(* IEC 61131-3 sources: AXOpen/src/components.drives/ctrl/src/AxoDrives (part 3) *)

            IF Enable THEN
                AxoReadActualPosition_Task.SwitchOn();
            ELSE
                AxoReadActualPosition_Task.SwitchOff();
                // THIS.MC_ReadActualPosition(AxisRef, FALSE);
            END_IF;

            Valid       := AxoReadActualPosition_Valid;
            Busy        :=  AxoReadActualPosition_Busy;
            Error       :=  AxoReadActualPosition_Error;
            ErrorID     :=  AxoReadActualPosition_ErrorID;
            Position    := AxoReadActualPosition_Value;

            AxoReadActualPosition  := AxoReadActualPosition_Task;
        END_METHOD

        ///<summary>
        /// This method returns the value of the actual velocity as long as ‘Enable’ is set. ‘Valid’ is true when the
        /// dataoutput ‘Velocity’ is valid. If ‘Enable’ is Reset, the data loses its validity, and all outputs are reset,
        /// no matter if new data is available.
        ///<summary>
        METHOD PUBLIC AxoReadActualVelocity    : IAxoToggleTask
            VAR_INPUT
                Enable          :   BOOL;                       //  Get the value of the parameter continuously while enabled
            END_VAR
            VAR_OUTPUT
                Valid           :   BOOL;                       //  A valid output is available at the method
                Busy            :   BOOL;                       //  The method is not finished and new output values are to be expected
                Error           :   BOOL;                       //  Signals that an error has occurred within the method
                ErrorID         :   DINT;                       //  Error identification
                Velocity        :   LREAL;                      //  The value of the actual velocity (in axis’ unit [u/s])
            END_VAR

            IF Enable THEN
                AxoReadActualVelocity_Task.SwitchOn();
            ELSE
                AxoReadActualVelocity_Task.SwitchOff();
                // THIS.MC_ReadActualVelocity(AxisRef, FALSE);
            END_IF;

            Valid       :=  AxoReadActualVelocity_Valid;
            Busy        :=  AxoReadActualVelocity_Busy;
            Error       :=  AxoReadActualVelocity_Error;
            ErrorID     :=  AxoReadActualVelocity_ErrorID;
            Velocity    :=  AxoReadActualVelocity_Value;

            AxoReadActualVelocity  := AxoReadActualVelocity_Task;
        END_METHOD

        ///<summary>
        /// This method returns the value of the actual torque or force as long as ‘Enable’ is set. ‘Valid’ is true when the
        /// data-output ‘Torque’ is valid. If ‘Enable’ is Reset, the data loses its validity, and ‘Valid’ is also reset,
        /// no matter if new data is available.
        ///<summary>
        METHOD PUBLIC AxoReadActualTorque  : IAxoToggleTask
            VAR_INPUT
                Enable          :   BOOL;                       //  Get the value of the parameter continuously while enabled
            END_VAR
            VAR_OUTPUT
                Valid           :   BOOL;                       //  A valid output is available at the method
                Busy            :   BOOL;                       //  The method is not finished and new output values are to be expected
                Error           :   BOOL;                       //  Signals that an error has occurred within the method
                ErrorID         :   DINT;                       //  Error identification
                Torque          :   LREAL;                      //  The value of the actual torque or force (in technical units)
            END_VAR

            IF Enable THEN
                AxoReadActualTorque_Task.SwitchOn();
            ELSE
                AxoReadActualTorque_Task.SwitchOff();
                // THIS.MC_ReadActualTorque(AxisRef, FALSE);
            END_IF;

            Valid   :=  AxoReadActualTorque_Valid;
            Busy    :=  AxoReadActualTorque_Busy;
            Error   :=  AxoReadActualTorque_Error;
            ErrorID :=  AxoReadActualTorque_ErrorID;
            Torque  :=  AxoReadActualTorque_Value;

            AxoReadActualTorque  := AxoReadActualTorque_Task;
        END_METHOD

        ///<summary>
        /// This method returns in detail the status of the state diagram of the axis
        ///<summary>
        METHOD PUBLIC AxoReadStatus    : IAxoToggleTask
            VAR_INPUT
                Enable          :   BOOL;                       //  Get the value of the parameter continuously while enabled
            END_VAR
            VAR_OUTPUT
                Valid           :   BOOL;                       //  A valid output is available at the method
                Busy            :   BOOL;                       //  The method is not finished and new output values are to be expected
                Error           :   BOOL;                       //  Signals that an error has occurred within the method
                ErrorID         :   DINT;                       //  Error identification
                ErrorStop       :   BOOL;                       //  See state diagram
                Disabled        :   BOOL;                       //  See state diagram
                Stopping        :   BOOL;                       //  See state diagram
                Homing          :   BOOL;                       //  See state diagram
                Standstill      :   BOOL;                       //  See state diagram
                DiscreteMotion  :   BOOL;                       //  See state diagram
                ContinuousMotion:   BOOL;                       //  See state diagram
                SynchronizedMotion: BOOL;                       //  See state diagram
            END_VAR

            IF Enable THEN
                AxoReadStatus_Task.SwitchOn();
            ELSE
                AxoReadStatus_Task.SwitchOff();
                // THIS.MC_ReadStatus(AxisRef, FALSE);
            END_IF;

            Valid               :=  AxoReadStatus_Valid;
            Busy                :=  AxoReadStatus_Busy;
            Error               :=  AxoReadStatus_Error;
            ErrorID             :=  AxoReadStatus_ErrorID;
            ErrorStop           :=  AxoReadStatus_ErrorStop;
            Disabled            :=  AxoReadStatus_Disabled;
            Stopping            :=  AxoReadStatus_Stopping;
            Homing              :=  AxoReadStatus_Homing;
            Standstill          :=  AxoReadStatus_Standstill;
            DiscreteMotion      :=  AxoReadStatus_DiscreteMotion;
            ContinuousMotion    :=  AxoReadStatus_ContinuousMotion;
            SynchronizedMotion  :=  AxoReadStatus_SynchronizedMotion;

            AxoReadStatus  := AxoReadStatus_Task;
        END_METHOD

        ///<summary>
        /// This method returns in detail the status of the axis with respect to the motion currently in progress.
        ///<summary>
        METHOD PUBLIC AxoReadMotionState   : IAxoToggleTask
            VAR_INPUT
                Enable          :   BOOL;                       //  Get the value of the parameter continuously while enabled
                Source          :   AXOpen.Components.Abstractions.Drives.eAxoSource;                 //  Defines the source of the relevant data: CommandedValue;SetValue, ActualValue.
            END_VAR
            VAR_OUTPUT
                Valid           :   BOOL;                       //  A valid output is available at the method
                Busy            :   BOOL;                       //  The method is not finished and new output values are to be expected
                Error           :   BOOL;                       //  Signals that an error has occurred within the method
                ErrorID         :   DINT;                       //  Error identification
                ConstantVelocity:   BOOL;                       //  Velocity is constant. Velocity may be 0. For the actual value a window is applicable (window is vendor specific)
                Accelerating    :   BOOL;                       //  Increasing the absolute value of the velocity
                Decelerating    :   BOOL;                       //  Decreasing the absolute value of the velocity
                DirectionPositive:  BOOL;                       //  Signals that the position is increasing
                DirectionNegative:  BOOL;                       //  Signals that the position is decreasing
            END_VAR

            IF Enable THEN
                AxoReadMotionState_Task.SwitchOn();
            ELSE
                AxoReadMotionState_Task.SwitchOff();
                // THIS.MC_ReadMotionState(AxisRef, FALSE);
            END_IF;

            Valid               :=  AxoReadMotionState_Valid;
            Busy                :=  AxoReadMotionState_Busy;
            Error               :=  AxoReadMotionState_Error;
            ErrorID             :=  AxoReadMotionState_ErrorID;
            ConstantVelocity    :=  AxoReadMotionState_ConstantVelocity;
            Accelerating        :=  AxoReadMotionState_Accelerating;
            Decelerating        :=  AxoReadMotionState_Decelerating;
            DirectionPositive   :=  AxoReadMotionState_DirectionPositive;
            DirectionNegative   :=  AxoReadMotionState_DirectionNegative;

            AxoReadMotionState  := AxoReadMotionState_Task;
        END_METHOD

        ///<summary>
        /// This method reads information concerning an axis, like modes, inputs directly related to the axis,
        /// and certain status information.
        ///<summary>
        METHOD PUBLIC AxoReadAxisInfo  : IAxoToggleTask
            VAR_INPUT
                Enable          :   BOOL;                       //  Get the value of the parameter continuously while enabled
            END_VAR
            VAR_OUTPUT
                Valid           :   BOOL;                       //  A valid output is available at the method
                Busy            :   BOOL;                       //  The method is not finished and new output values are to be expected
                Error           :   BOOL;                       //  Signals that an error has occurred within the method
                ErrorID         :   DINT;                       //  Error identification
                HomeAbsSwitch   :   BOOL;                       //  Digital home switch input is active
                LimitSwitchPos  :   BOOL;                       //  Positive hardware end switch is active
                LimitSwitchNeg  :   BOOL;                       //  Negative hardware end switch is active
                Simulation      :   BOOL;                       //  Axis is in simulation mode (e.g. motor is simulated)
                CommunicationReady: BOOL;                       //  “Network” is initialized and ready for communication
                ReadyForPowerOn :   BOOL;                       //  Drive is ready to be enabled (power on)
                PowerOn         :   BOOL;                       //  If TRUE shows that the power stage is switched ON
                IsHomed         :   BOOL;                       //  The absolute reference position is known for the axis (axis is homed)
                AxisWarning     :   BOOL;                       //  Warning(s) on the axis is present
            END_VAR

            IF Enable THEN
                AxoReadAxisInfo_Task.SwitchOn();
            ELSE
                AxoReadAxisInfo_Task.SwitchOff();
                // THIS.ReadAxisInfo(AxisRef, FALSE);
            END_IF;

            Valid               :=  AxoReadAxisInfo_Valid;
            Busy                :=  AxoReadAxisInfo_Busy;
            Error               :=  AxoReadAxisInfo_Error;
            ErrorID             :=  AxoReadAxisInfo_ErrorID;
            HomeAbsSwitch       :=  AxoReadAxisInfo_HomeAbsSwitch;
            LimitSwitchPos      :=  AxoReadAxisInfo_LimitSwitchPos;
            LimitSwitchNeg      :=  AxoReadAxisInfo_LimitSwitchNeg;
            Simulation          :=  AxoReadAxisInfo_Simulation;
            CommunicationReady  :=  AxoReadAxisInfo_CommunicationReady;
            ReadyForPowerOn     :=  AxoReadAxisInfo_ReadyForPowerOn;
            PowerOn             :=  AxoReadAxisInfo_PowerOn;
            IsHomed             :=  AxoReadAxisInfo_IsHomed;
            AxisWarning         :=  AxoReadAxisInfo_AxisWarning;

            AxoReadAxisInfo  := AxoReadAxisInfo_Task;
        END_METHOD

        ///<summary>
        /// This method presents general axis errors not relating to the methods.
        /// (for instance axis errors, drive errors, communication errors)
        ///<summary>
        METHOD PUBLIC AxoReadAxisError : IAxoToggleTask
            VAR_INPUT
                Enable          :   BOOL;                       //  Get the value of the parameter continuously while enabled
            END_VAR
            VAR_OUTPUT
                Valid           :   BOOL;                       //  A valid output is available at the method
                Busy            :   BOOL;                       //  The method is not finished and new output values are to be expected
                Error           :   BOOL;                       //  Signals that an error has occurred within the method
                ErrorID         :   DINT;                       //  Error identification
                AxisErrorID     :   DWORD;                      //  The value of the axis error. These values are vendor specific
            END_VAR

            IF Enable THEN
                AxoReadAxisError_Task.SwitchOn();
            ELSE
                AxoReadAxisError_Task.SwitchOff();
                // THIS.MC_ReadAxisError(FALSE);
            END_IF;

            Valid           :=  AxoReadAxisError_Valid;
            Busy            :=  AxoReadAxisError_Busy;
            Error           :=  AxoReadAxisError_Error;
            ErrorID         :=  AxoReadAxisError_ErrorID;
            AxisErrorID     :=  AxoReadAxisError_AxisErrorID;

            AxoReadAxisError  := AxoReadAxisError_Task;
        END_METHOD

        ///<summary>
        /// This method makes the transition from the state ‘ErrorStop’ to ‘Standstill’ or ‘Disabled’ by resetting all
        /// internal axis-related errors – it does not affect the output of the other methods.
        ///<summary>
        METHOD PUBLIC AxoReset : IAxoTaskState
            VAR_OUTPUT
                Done            :   BOOL;                       //  ‘Standstill’ or ‘Disabled’ state is reached
                Busy            :   BOOL;                       //  The method is not finished and new output values are to be expected
                Error           :   BOOL;                       //  Signals that an error has occurred within the method
                ErrorID         :   DINT;                       //  Error identification
            END_VAR

            Done        :=  AxoReset_Done;
            Busy        :=  AxoReset_Busy;
            Error       :=  AxoReset_Error;
            ErrorID     :=  AxoReset_ErrorID;

            AxoReset    := AxoReset_Task.Invoke(THIS);
        END_METHOD

        ///<summary>
        /// Ensures reading the hardware input data into the AxisRef data structure
        /// This vendor specific method must be overridden in derived class.
        ///</summary>
        METHOD PROTECTED ABSTRACT UpdateInputs : BOOL
            VAR_INPUT
                AxisRef         :   AXOpen.Components.Abstractions.Drives.IAxoAxisReference;
            END_VAR
        END_METHOD

        ///<summary>
        /// Ensures writing the AxisRef data structure into the hardware output data
        /// This vendor specific method must be overridden in derived class.
        ///</summary>
        METHOD PROTECTED ABSTRACT UpdateOutputs : BOOL
            VAR_INPUT
                AxisRef         :   AXOpen.Components.Abstractions.Drives.IAxoAxisReference;
            END_VAR
        END_METHOD

        ///<summary>
        /// This method controls the power stage (On or Off).
        /// This vendor specific method must be overridden in derived class.
        ///</summary>
        METHOD PUBLIC ABSTRACT MC_Power
            VAR_INPUT
                AxisRef         :   AXOpen.Components.Abstractions.Drives.IAxoAxisReference;
                Enable          :   BOOL;                       //  As long as ‘Enable’ is true, power is being enabled.
            END_VAR
            VAR_OUTPUT
                Status          :   BOOL;                       //  Effective state of the power stage
                Valid           :   BOOL;                       //  If true, a valid set of outputs is available at the method
                Error           :   BOOL;                       //  Signals that an error has occurred within the method
                ErrorID         :   DINT;                       //  Error identification
            END_VAR
        END_METHOD

        ///<summary>
        /// This method commands the axis to perform the «search home» sequence. The details of this sequence are
        /// manufacturer dependent and can be set by the axis’ parameters. The ‘Position’ input is used to set the absolute
        /// position when reference signal is detected. This method completes at ‘Standstill’ if it was started in ‘Standstill’.
        /// This vendor specific method must be overridden in the derived class.
        ///</summary>
        METHOD PUBLIC ABSTRACT MC_Home
            VAR_INPUT
                AxisRef         :   AXOpen.Components.Abstractions.Drives.IAxoAxisReference;
                Execute         :   BOOL;                       //  Start the motion at rising edge
                Position        :   LREAL;                      //  Absolute position when the reference signal is detected
                HommingMode     :   INT;                        //  Required homming mode
                Velocity        :   LREAL;                      //  Value of the maximum ‘Velocity’ (not necessarily reached) [u/s].
                Acceleration    :   LREAL;                      //  Value of the ‘Acceleration’ (always positive) (increasing energy of the motor) [u/s2]
                Deceleration    :   LREAL;                      //  Value of the ‘Deceleration’ (always positive) (decreasing energy of the motor) [u/s2]
            END_VAR
            VAR_OUTPUT
                Done            :   BOOL;                       // Reference known and set sucessfully
                Busy            :   BOOL;                       // The method is not finished and new output values are to be expected
                Active          :   BOOL;                       // Indicates that the method has control on the axis
                CommandAborted  :   BOOL;                       // ‘Command’ is aborted by another command
                Error           :   BOOL;                       // Signals that an error has occurred within the method
                ErrorID         :   DINT;                       // Error identification
             END_VAR
        END_METHOD

        ///<summary>
        /// This method commands a controlled motion stop and transfers the axis to the state ‘Stopping’. It aborts any
        /// ongoing method execution. While the axis is in state ‘Stopping’, no other method can perform any motion on the
        /// same axis.
        /// This vendor specific method must be overridden in the derived class.
        ///</summary>
        METHOD PUBLIC ABSTRACT MC_Stop
            VAR_INPUT
                AxisRef         :   AXOpen.Components.Abstractions.Drives.IAxoAxisReference;
                Execute         :   BOOL;                       //  Start the action at rising edge
                Deceleration    :   LREAL;                      //  Value of the ‘Deceleration’ [u/s2]
                Jerk            :   LREAL;                      //  Value of the ‘Jerk’ [u/s3]
            END_VAR
            VAR_OUTPUT
                Done            :   BOOL;                       // Zero velocity reached
                Busy            :   BOOL;                       // The method is not finished and new output values are to be expected
                Active          :   BOOL;                       // Indicates that the method has control on the axis
                CommandAborted  :   BOOL;                       // ‘Command’ is aborted by switching off power (only possibility to abort)
                Error           :   BOOL;                       // Signals that an error has occurred within the method
                ErrorID         :   DINT;                       // Error identification
             END_VAR
        END_METHOD

        ///<summary>
        /// This method commands a controlled motion stop. The axis is moved to the state ‘DiscreteMotion’, until the
        /// velocity is zero. With the ‘Done’ output set, the state is transferred to ‘Standstill’.
        /// This vendor specific method must be overridden in the derived class.
        ///</summary>
        METHOD PUBLIC ABSTRACT MC_Halt
            VAR_INPUT
                AxisRef         :   AXOpen.Components.Abstractions.Drives.IAxoAxisReference;
                Execute         :   BOOL;                       //  Start the action at rising edge
                Deceleration    :   LREAL;                      //  Value of the ‘Deceleration’ [u/s2]
                Jerk            :   LREAL;                      //  Value of the ‘Jerk’ [u/s3]
            END_VAR
            VAR_OUTPUT
                Done            :   BOOL;                       // Zero velocity reached
                Busy            :   BOOL;                       // The method is not finished and new output values are to be expected
                Active          :   BOOL;                       // Indicates that the method has control on the axis
                CommandAborted  :   BOOL;                       // ‘Command’ is aborted by switching off power (only possibility to abort)
                Error           :   BOOL;                       // Signals that an error has occurred within the method
                ErrorID         :   DINT;                       // Error identification
             END_VAR
        END_METHOD

        ///<summary>
        /// This method commands a controlled motion to a specified absolute position.
        /// This vendor specific method must be overridden in the derived class.
        ///<summary>
        METHOD PUBLIC ABSTRACT MC_MoveAbsolute
            VAR_INPUT
                AxisRef         :   AXOpen.Components.Abstractions.Drives.IAxoAxisReference;
                Execute         :   BOOL;                       //  Start the motion at rising edge
                ContinuousUpdate:   BOOL;                       //  Activate ‘ContinuousUpdate’ - target parameters should be changed during movement
                Position        :   LREAL;                      //  Commanded ‘Position’ for the motion (in technical unit [u]) (negative or positive)
                Velocity        :   LREAL;                      //  Value of the maximum ‘Velocity’ (not necessarily reached) [u/s].
                Acceleration    :   LREAL;                      //  Value of the ‘Acceleration’ (always positive) (increasing energy of the motor) [u/s2]
                Deceleration    :   LREAL;                      //  Value of the ‘Deceleration’ (always positive) (decreasing energy of the motor) [u/s2]
                Jerk            :   LREAL;                      //  Value of the ‘Jerk’ [u/s3]
                Direction       :   AXOpen.Components.Abstractions.Drives.eAxoDriveDirection;         //  Enum type (1-of-4 values: PositiveDirection, ShortestWay, NegativeDirection, CurrentDirection)
            END_VAR
            VAR_OUTPUT
                Done            :   BOOL;                       // Commanded position finally reached
                Busy            :   BOOL;                       // The method is not finished and new output values are to be expected
                Active          :   BOOL;                       // Indicates that the method has control on the axis
                CommandAborted  :   BOOL;                       // ‘Command’ is aborted by another command
                Error           :   BOOL;                       // Signals that an error has occurred within the method
                ErrorID         :   DINT;                       // Error identification
             END_VAR
        END_METHOD

        ///<summary>
        /// This method  commands a controlled motion of a specified distance relative to the set position at the time of the execution.
        /// This vendor specific method must be overridden in the derived class.
        ///<summary>
        METHOD PUBLIC ABSTRACT MC_MoveRelative
            VAR_INPUT
                AxisRef         :   AXOpen.Components.Abstractions.Drives.IAxoAxisReference;
                Execute         :   BOOL;                       //  Start the motion at rising edge
                ContinuousUpdate:   BOOL;                       //  Activate ‘ContinuousUpdate’ - target parameters should be changed during movement
                Distance        :   LREAL;                      //  Relative distance for the motion (in technical unit [u]
                Velocity        :   LREAL;                      //  Value of the maximum ‘Velocity’ (not necessarily reached) [u/s].
                Acceleration    :   LREAL;                      //  Value of the ‘Acceleration’ (always positive) (increasing energy of the motor) [u/s2]
                Deceleration    :   LREAL;                      //  Value of the ‘Deceleration’ (always positive) (decreasing energy of the motor) [u/s2]
                Jerk            :   LREAL;                      //  Value of the ‘Jerk’ [u/s3]
            END_VAR
            VAR_OUTPUT
                Done            :   BOOL;                       // Commanded distance reached
                Busy            :   BOOL;                       // The method is not finished and new output values are to be expected
                Active          :   BOOL;                       // Indicates that the method has control on the axis
                CommandAborted  :   BOOL;                       // ‘Command’ is aborted by another command
                Error           :   BOOL;                       // Signals that an error has occurred within the method
                ErrorID         :   DINT;                       // Error identification
             END_VAR
        END_METHOD

        ///<summary>
        /// This method commands a controlled motion of a specified relative distance additional to the most recent
        /// commanded position in the axis state ‘DiscreteMotion’. The most recent commanded position may be the result of a
        /// previous MC_MoveAdditive motion which was aborted. If the method is activated in the axis state ‘ContinuousMotion’, the
        /// specified relative distance is added to the set position at the time of the execution.
        /// This vendor specific method must be overridden in the derived class.
        ///<summary>
        METHOD PUBLIC ABSTRACT MC_MoveAdditive
            VAR_INPUT
                AxisRef         :   AXOpen.Components.Abstractions.Drives.IAxoAxisReference;
                Execute         :   BOOL;                       //  Start the motion at rising edge
                ContinuousUpdate:   BOOL;                       //  Activate ‘ContinuousUpdate’ - target parameters should be changed during movement
                Distance        :   LREAL;                      //  Relative distance for the motion (in technical unit [u]
                Velocity        :   LREAL;                      //  Value of the maximum ‘Velocity’ (not necessarily reached) [u/s].
                Acceleration    :   LREAL;                      //  Value of the ‘Acceleration’ (always positive) (increasing energy of the motor) [u/s2]
                Deceleration    :   LREAL;                      //  Value of the ‘Deceleration’ (always positive) (decreasing energy of the motor) [u/s2]
                Jerk            :   LREAL;                      //  Value of the ‘Jerk’ [u/s3]
            END_VAR
            VAR_OUTPUT
                Done            :   BOOL;                       // Commanded distance reached
                Busy            :   BOOL;                       // The method is not finished and new output values are to be expected
                Active          :   BOOL;                       // Indicates that the method has control on the axis
                CommandAborted  :   BOOL;                       // ‘Command’ is aborted by another command
                Error           :   BOOL;                       // Signals that an error has occurred within the method
                ErrorID         :   DINT;                       // Error identification
             END_VAR
        END_METHOD

        ///<summary>
        /// This method commands a never ending controlled motion at a specified velocity.
        /// This vendor specific method must be overridden in the derived class.
        ///<summary>
        METHOD PUBLIC ABSTRACT MC_MoveVelocity
            VAR_INPUT
                AxisRef         :   AXOpen.Components.Abstractions.Drives.IAxoAxisReference;
                Execute         :   BOOL;                       //  Start the motion at rising edge
                ContinuousUpdate:   BOOL;                       //  Activate ‘ContinuousUpdate’ - target parameters should be changed during movement
                Velocity        :   LREAL;                      //  Value of the maximum velocity [u/s]. Can be a signed value.
                Acceleration    :   LREAL;                      //  Value of the ‘Acceleration’ (always positive) (increasing energy of the motor) [u/s2]
                Deceleration    :   LREAL;                      //  Value of the ‘Deceleration’ (always positive) (decreasing energy of the motor) [u/s2]
                Jerk            :   LREAL;                      //  Value of the ‘Jerk’ [u/s3]
                Direction       :   AXOpen.Components.Abstractions.Drives.eAxoDriveDirection;         //  Enum type (1-of-3 values: PositiveDirection, NegativeDirection, and CurrentDirection. Note: shortest way not applicable)
            END_VAR
            VAR_OUTPUT
                InVelocity      :   BOOL;                       // Commanded velocity reached
                Busy            :   BOOL;                       // The method is not finished and new output values are to be expected
                Active          :   BOOL;                       // Indicates that the method has control on the axis
                CommandAborted  :   BOOL;                       // ‘Command’ is aborted by another command
                Error           :   BOOL;                       // Signals that an error has occurred within the method
                ErrorID         :   DINT;                       // Error identification
             END_VAR
        END_METHOD

        ///<summary>
        /// This method continuously exerts a torque or force of the specified magnitude. This magnitude is
        /// approached using a defined ramp (‘TorqueRamp’), and the method sets the ‘InTorque’ output if the
        /// commanded torque level is reached. This method is applicable for force and torque. When there is no external
        /// load, force is applicable. Positive torque is in the positive direction of velocity.
        /// This vendor specific method must be overridden in the derived class.
        ///<summary>
        METHOD PUBLIC ABSTRACT MC_TorqueControl
            VAR_INPUT
                AxisRef         :   AXOpen.Components.Abstractions.Drives.IAxoAxisReference;
                Execute         :   BOOL;                       //  Start the motion at rising edge
                ContinuousUpdate:   BOOL;                       //  Activate ‘ContinuousUpdate’ - target parameters should be changed during movement
                Torque          :   LREAL;                      //  Value of the torque (Torque or force in technical unit [u])
                TorqueRamp      :   LREAL;                      //  The maximum time derivative of the set value of the torque or force (in technical unit per sec. [u/s])
                PositionLimit   :   LREAL;                      //  Position limit.
                Velocity        :   LREAL;                      //  Absolute value of the maximum velocity.
                Acceleration    :   LREAL;                      //  Value of the maximum acceleration (acceleration is applicable with same sign of torque and velocity)
                Deceleration    :   LREAL;                      //  Value of the maximum deceleration (deceleration is applicable with opposite signs of torque and velocity)
                Jerk            :   LREAL;                      //  Value of the maximum jerk
                Direction       :   AXOpen.Components.Abstractions.Drives.eAxoDriveDirection;         //  Enum type (1 of 2 values: PositiveDirection, NegativeDirection or CurrentDirection). Specifies the direction of the torque. (Note: Torque input can be signed value).
            END_VAR
            VAR_OUTPUT
                InTorque        :   BOOL;                       //  Setpoint value of torque or force equals the commandedvalue
                Busy            :   BOOL;                       //  The method is not finished and new output values are to be expected
                Active          :   BOOL;                       //  Indicates that the method has control on the axis
                CommandAborted  :   BOOL;                       //  ‘Command’ is aborted by another command
                Error           :   BOOL;                       //  Signals that an error has occurred within the method
                ErrorID         :   DINT;                       //  Error identification
            END_VAR
        END_METHOD

        ///<summary>
        /// This method shifts the coordinate system of an axis by manipulating both the set-point position as well as the
        /// actual position of an axis with the same value without any movement caused. (Re-calibration with same following error).
        /// This can be used for instance for a reference situation. This method can also be used during motion without changing
        /// the commanded position, which is now positioned in the shifted coordinate system.
        /// This vendor specific method must be overridden in the derived class.
        ///<summary>
        METHOD PUBLIC ABSTRACT MC_SetPosition
            VAR_INPUT
                AxisRef         :   AXOpen.Components.Abstractions.Drives.IAxoAxisReference;
                Execute         :   BOOL;                       //  Start setting position in axis
                Position        :   LREAL;                      //  Position unit [u] (Means ‘Distance’ if ‘Relative’= TRUE)
                Relative        :   BOOL;                       //  ‘Relative’ distance if True, ‘Absolute’ position if False (= Default)
                ExecutionMode   :   AXOpen.Components.Abstractions.Drives.eAxoExecutionMode;          //  Defines the chronological sequence of the method.
            END_VAR
            VAR_OUTPUT
                Done            :   BOOL;                       //  ‘Position’ has new value
                Busy            :   BOOL;                       //  The method is not finished and new output values are to be expected
                Error           :   BOOL;                       //  Signals that an error has occurred within the method
                ErrorID         :   DINT;                       //  Error identification
            END_VAR
        END_METHOD

        ///<summary>
        /// This method sets the values of override for the whole axis, and all functions that are working on that axis. The override
        /// parameters contribute as a factor to the calculation of the commanded velocity, acceleration and jerk of the motion.
        /// This vendor specific method must be overridden in the derived class.
        ///<summary>
        METHOD PUBLIC ABSTRACT MC_SetOverride
            VAR_INPUT
                AxisRef         :   AXOpen.Components.Abstractions.Drives.IAxoAxisReference;
                Enable          :   BOOL;                       //  If SET, it writes the value of the override factor continuously. If RESET it should keep the last value.
                VelocityFactor  :   LREAL;                      //  New override factor for the velocity
                AccelerationFactor:   LREAL;                      //  New override factor for the acceleration/deceleration
                JerkFactor      :   LREAL;                      //  New override factor for the jer
            END_VAR
            VAR_OUTPUT
                Enabled         :   BOOL;                       //  Signals that the override factor(s) is (are) set successfully
                Busy            :   BOOL;                       //  The method is not finished and new output values are to be expected
                Error           :   BOOL;                       //  Signals that an error has occurred within the method
                ErrorID         :   DINT;                       //  Error identification
            END_VAR
        END_METHOD

        ///<summary>
        /// This method returns the value of a vendor specific parameter. The returned Value has to be converted to Real
        /// if necessary. If not possible, the vendor has to supply a vendor specific method to read the parameter.
        /// This vendor specific method must be overridden in the derived class.
        ///<summary>
        METHOD PUBLIC ABSTRACT MC_ReadParameter
            VAR_INPUT
                AxisRef         :   AXOpen.Components.Abstractions.Drives.IAxoAxisReference;
                Enable          :   BOOL;                       //  Get the value of the parameter continuously while enabled
                ParameterNumber :   DINT;                       //  Number of the parameter. One can also use symbolic parameter names which are declared as VAR CONST.
            END_VAR
            VAR_OUTPUT
                Valid           :   BOOL;                       //  A valid output is available at the method
                Busy            :   BOOL;                       //  The method is not finished and new output values are to be expected
                Error           :   BOOL;                       //  Signals that an error has occurred within the method
                ErrorID         :   DINT;                       //  Error identification
                Value           :   LINT;                       //  Value of the specified parameter in the datatype, as specified by the vendor
            END_VAR
        END_METHOD

        ///<summary>
        /// This method returns the value of a vendor specific parameter with datatype REAL.
        /// This vendor specific method must be overridden in the derived class.
        ///<summary>
        METHOD PUBLIC ABSTRACT MC_ReadRealParameter
            VAR_INPUT
                AxisRef         :   AXOpen.Components.Abstractions.Drives.IAxoAxisReference;
                Enable          :   BOOL;                       //  Get the value of the parameter continuously while enabled
                ParameterNumber :   DINT;                       //  Number of the parameter. One can also use symbolic parameter names which are declared as VAR CONST.
            END_VAR
            VAR_OUTPUT
                Valid           :   BOOL;                       //  A valid output is available at the method
                Busy            :   BOOL;                       //  The method is not finished and new output values are to be expected
                Error           :   BOOL;                       //  Signals that an error has occurred within the method
                ErrorID         :   DINT;                       //  Error identification
                Value           :   REAL;                       //  Value of the specified parameter in the datatype, as specified by the vendor
            END_VAR
        END_METHOD

        ///<summary>
        /// This method returns the value of a vendor specific parameter with datatype BOOL.
        /// This vendor specific method must be overridden in the derived class.
        ///<summary>
        METHOD PUBLIC ABSTRACT MC_ReadBoolParameter
            VAR_INPUT
                AxisRef         :   AXOpen.Components.Abstractions.Drives.IAxoAxisReference;
                Enable          :   BOOL;                       //  Get the value of the parameter continuously while enabled
                ParameterNumber :   DINT;                       //  Number of the parameter. One can also use symbolic parameter names which are declared as VAR CONST.
            END_VAR
            VAR_OUTPUT
                Valid           :   BOOL;                       //  A valid output is available at the method
                Busy            :   BOOL;                       //  The method is not finished and new output values are to be expected
                Error           :   BOOL;                       //  Signals that an error has occurred within the method
                ErrorID         :   DINT;                       //  Error identification
                Value           :   BOOL;                       //  Value of the specified parameter in the datatype, as specified by the vendor
            END_VAR
        END_METHOD

        ///<summary>
        /// This method modifies the value of a vendor specific parameter.
        /// This vendor specific method must be overridden in the derived class.
        ///<summary>
        METHOD PUBLIC ABSTRACT MC_WriteParameter
            VAR_INPUT
                AxisRef         :   AXOpen.Components.Abstractions.Drives.IAxoAxisReference;
                Execute         :   BOOL;                       //  Write the value of the parameter at rising edge
                ParameterNumber :   DINT;                       //  Number of the parameter (correspondence between number andparameter is specified in the table above)
                Value           :   LINT;                       //  New value of the specified parameter
                ExecutionMode   :   AXOpen.Components.Abstractions.Drives.eAxoExecutionMode;          //  Defines the chronological sequence of the method.
            END_VAR
            VAR_OUTPUT
                Done            :   BOOL;                       //  Parameter successfully written
                Busy            :   BOOL;                       //  The method is not finished and new output values are to be expected.
                Error           :   BOOL;                       //  Signals that an error has occurred within the method
                ErrorID         :   DINT;                       //  Error identification
            END_VAR
        END_METHOD

        ///<summary>
        /// This method modifies the value of a vendor specific parameter of type REAL.
        /// This vendor specific method must be overridden in the derived class.
        ///<summary>
        METHOD PUBLIC ABSTRACT MC_WriteRealParameter
            VAR_INPUT
                AxisRef         :   AXOpen.Components.Abstractions.Drives.IAxoAxisReference;
                Execute         :   BOOL;                       //  Write the value of the parameter at rising edge
                ParameterNumber :   DINT;                       //  Number of the parameter (correspondence between number andparameter is specified in the table above)
                Value           :   REAL;                       //  New value of the specified parameter
                ExecutionMode   :   AXOpen.Components.Abstractions.Drives.eAxoExecutionMode;          //  Defines the chronological sequence of the method.
            END_VAR
            VAR_OUTPUT
                Done            :   BOOL;                       //  Parameter successfully written
                Busy            :   BOOL;                       //  The method is not finished and new output values are to be expected.
                Error           :   BOOL;                       //  Signals that an error has occurred within the method
                ErrorID         :   DINT;                       //  Error identification
            END_VAR
        END_METHOD

        ///<summary>
        /// This method modifies the value of a vendor specific parameter of type BOOL.
        /// This vendor specific method must be overridden in the derived class.
        ///<summary>
        METHOD PUBLIC ABSTRACT MC_WriteBoolParameter
            VAR_INPUT
                AxisRef         :   AXOpen.Components.Abstractions.Drives.IAxoAxisReference;
                Execute         :   BOOL;                       //  Write the value of the parameter at rising edge
                ParameterNumber :   DINT;                       //  Number of the parameter (correspondence between number andparameter is specified in the table above)
                Value           :   BOOL;                       //  New value of the specified parameter
                ExecutionMode   :   AXOpen.Components.Abstractions.Drives.eAxoExecutionMode;          //  Defines the chronological sequence of the method.
            END_VAR
            VAR_OUTPUT
                Done            :   BOOL;                       //  Parameter successfully written
                Busy            :   BOOL;                       //  The method is not finished and new output values are to be expected.
                Error           :   BOOL;                       //  Signals that an error has occurred within the method
                ErrorID         :   DINT;                       //  Error identification
            END_VAR
        END_METHOD

        ///<summary>
        /// This method gives access to the value of the input, referenced by the datatype MC_INPUT_REF.
        /// It provides the value of the referenced input (BOOL).
        /// This vendor specific method must be overridden in the derived class.
        ///<summary>
        METHOD PUBLIC ABSTRACT MC_ReadDigitalInput
            VAR_INPUT
                AxisRef         :   AXOpen.Components.Abstractions.Drives.IAxoAxisReference;
                Enable          :   BOOL;                       //  Get the value of the selected input signal continuously while enabled
                InputNumber     :   INT;                        //  Selects the input. Can be part of MC_INPUT_REF, if only one single input is referenced.
            END_VAR
            VAR_OUTPUT
                Valid           :   BOOL;                       //  A valid output is available at the method
                Busy            :   BOOL;                       //  The method is not finished and new output values are to be expected
                Error           :   BOOL;                       //  Signals that an error has occurred within the method
                ErrorID         :   DINT;                       //  Error identification
                Value           :   BOOL;                       //  The value of the selected input signal
            END_VAR
        END_METHOD

        ///<summary>
        /// This method provides access to the value of a digital output, referenced by the datatype MC_OUTPUT_REF.
        /// It provides the value of the referenced output (BOOL).
        /// This vendor specific method must be overridden in the derived class.
        ///<summary>
        METHOD PUBLIC ABSTRACT MC_ReadDigitalOutput
            VAR_INPUT
                AxisRef         :   AXOpen.Components.Abstractions.Drives.IAxoAxisReference;
                Enable          :   BOOL;                       //  Get the value of the selected output signal continuously while enabled
                OutputNumber    :   INT;                        //  Selects the output. Can be part of MC_OUTPUT_REF, if only one single output is referenced.
            END_VAR
            VAR_OUTPUT
                Valid           :   BOOL;                       //  A valid output is available at the method
                Busy            :   BOOL;                       //  The method is not finished and new output values are to be expected
                Error           :   BOOL;                       //  Signals that an error has occurred within the method
                ErrorID         :   DINT;                       //  Error identification
                Value           :   BOOL;                       //  The value of the selected output signal
            END_VAR
        END_METHOD

        ///<summary>
        /// This method writes a value to the output referenced by the argument ‘Output’ once (with rising edge of Execute)
        /// This vendor specific method must be overridden in the derived class.
        ///<summary>
        METHOD PUBLIC ABSTRACT MC_WriteDigitalOutput
            VAR_INPUT
                AxisRef         :   AXOpen.Components.Abstractions.Drives.IAxoAxisReference;
                Execute         :   BOOL;                       //  Write the value of the selected output
                OutputNumber    :   INT;                        //  Selects the output. Can be part of MC_OUTPUT_REF, if only one single output is referenced.
                Value           :   BOOL;                       //  The value of the selected output signal
                ExecutionMode   :   AXOpen.Components.Abstractions.Drives.eAxoExecutionMode;          //  Defines the chronological sequence of the method.
            END_VAR
            VAR_OUTPUT
                Done            :   BOOL;                       //  Writing of the output signal value is done
                Busy            :   BOOL;                       //  The method is not finished and new output values are to be expected.
                Error           :   BOOL;                       //  Signals that an error has occurred within the method
                ErrorID         :   DINT;                       //  Error identification
            END_VAR
        END_METHOD

        ///<summary>
        /// This method returns the actual position.
        /// This vendor specific method must be overridden in the derived class.
        ///<summary>
        METHOD PUBLIC ABSTRACT MC_ReadActualPosition
            VAR_INPUT
                AxisRef         :   AXOpen.Components.Abstractions.Drives.IAxoAxisReference;
                Enable          :   BOOL;                       //  Get the value of the parameter continuously while enabled
            END_VAR
            VAR_OUTPUT
                Valid           :   BOOL;                       //  A valid output is available at the method
                Busy            :   BOOL;                       //  The method is not finished and new output values are to be expected
                Error           :   BOOL;                       //  Signals that an error has occurred within the method
                ErrorID         :   DINT;                       //  Error identification
                Position        :   LREAL;                       //  New absolute position (in axis’ unit [u])
            END_VAR
        END_METHOD

        ///<summary>
        /// This method returns the value of the actual velocity as long as ‘Enable’ is set. ‘Valid’ is true when the
        /// dataoutput ‘Velocity’ is valid. If ‘Enable’ is Reset, the data loses its validity, and all outputs are reset,
        /// no matter if new data is available.
        /// This vendor specific method must be overridden in the derived class.
        ///<summary>
        METHOD PUBLIC ABSTRACT MC_ReadActualVelocity
            VAR_INPUT
                AxisRef         :   AXOpen.Components.Abstractions.Drives.IAxoAxisReference;
                Enable          :   BOOL;                       //  Get the value of the parameter continuously while enabled
            END_VAR
            VAR_OUTPUT
                Valid           :   BOOL;                       //  A valid output is available at the method
                Busy            :   BOOL;                       //  The method is not finished and new output values are to be expected
                Error           :   BOOL;                       //  Signals that an error has occurred within the method
                ErrorID         :   DINT;                       //  Error identification
                Velocity        :   LREAL;                       //  The value of the actual velocity (in axis’ unit [u/s])
            END_VAR
        END_METHOD

        ///<summary>
        /// This method returns the value of the actual torque or force as long as ‘Enable’ is set. ‘Valid’ is true when the
        /// data-output ‘Torque’ is valid. If ‘Enable’ is Reset, the data loses its validity, and ‘Valid’ is also reset,
        /// no matter if new data is available.
        /// This vendor specific method must be overridden in the derived class.
        ///<summary>
        METHOD PUBLIC ABSTRACT MC_ReadActualTorque
            VAR_INPUT
                AxisRef         :   AXOpen.Components.Abstractions.Drives.IAxoAxisReference;
                Enable          :   BOOL;                       //  Get the value of the parameter continuously while enabled
            END_VAR
            VAR_OUTPUT
                Valid           :   BOOL;                       //  A valid output is available at the method
                Busy            :   BOOL;                       //  The method is not finished and new output values are to be expected
                Error           :   BOOL;                       //  Signals that an error has occurred within the method
                ErrorID         :   DINT;                       //  Error identification
                Torque          :   LREAL;                       //  The value of the actual torque or force (in technical units)
            END_VAR
        END_METHOD

        ///<summary>
        /// This method returns in detail the status of the state diagram of the axis
        /// This vendor specific method must be overridden in the derived class.
        ///<summary>
        METHOD PUBLIC ABSTRACT MC_ReadStatus
            VAR_INPUT
                AxisRef         :   AXOpen.Components.Abstractions.Drives.IAxoAxisReference;
                Enable          :   BOOL;                       //  Get the value of the parameter continuously while enabled
            END_VAR
            VAR_OUTPUT
                Valid           :   BOOL;                       //  A valid output is available at the method
                Busy            :   BOOL;                       //  The method is not finished and new output values are to be expected
                Error           :   BOOL;                       //  Signals that an error has occurred within the method
                ErrorID         :   DINT;                       //  Error identification
                ErrorStop       :   BOOL;                       //  See state diagram
                Disabled        :   BOOL;                       //  See state diagram
                Stopping        :   BOOL;                       //  See state diagram
                Homing          :   BOOL;                       //  See state diagram
                Standstill      :   BOOL;                       //  See state diagram
                DiscreteMotion  :   BOOL;                       //  See state diagram
                ContinuousMotion:   BOOL;                       //  See state diagram
                SynchronizedMotion: BOOL;                       //  See state diagram
            END_VAR
        END_METHOD

        ///<summary>
        /// This method returns in detail the status of the axis with respect to the motion currently in progress.
        /// This vendor specific method must be overridden in the derived class.
        ///<summary>
        METHOD PUBLIC ABSTRACT MC_ReadMotionState
            VAR_INPUT
                AxisRef         :   AXOpen.Components.Abstractions.Drives.IAxoAxisReference;
                Enable          :   BOOL;                       //  Get the value of the parameter continuously while enabled
                Source          :   AXOpen.Components.Abstractions.Drives.eAxoSource;                 //  Defines the source of the relevant data: CommandedValue;SetValue, ActualValue.
            END_VAR
            VAR_OUTPUT
                Valid           :   BOOL;                       //  A valid output is available at the method
                Busy            :   BOOL;                       //  The method is not finished and new output values are to be expected
                Error           :   BOOL;                       //  Signals that an error has occurred within the method
                ErrorID         :   DINT;                       //  Error identification
                ConstantVelocity:   BOOL;                       //  Velocity is constant. Velocity may be 0. For the actual value a window is applicable (window is vendor specific)
                Accelerating    :   BOOL;                       //  Increasing the absolute value of the velocity
                Decelerating    :   BOOL;                       //  Decreasing the absolute value of the velocity
                DirectionPositive:  BOOL;                       //  Signals that the position is increasing
                DirectionNegative:  BOOL;                       //  Signals that the position is decreasing
            END_VAR
        END_METHOD

        ///<summary>
        /// This method reads information concerning an axis, like modes, inputs directly related to the axis,
        /// and certain status information.
        /// This vendor specific method must be overridden in the derived class.
        ///<summary>
        METHOD PUBLIC ABSTRACT MC_ReadAxisInfo
            VAR_INPUT
                AxisRef         :   AXOpen.Components.Abstractions.Drives.IAxoAxisReference;
                Enable          :   BOOL;                       //  Get the value of the parameter continuously while enabled
            END_VAR
            VAR_OUTPUT
                Valid           :   BOOL;                       //  A valid output is available at the method
                Busy            :   BOOL;                       //  The method is not finished and new output values are to be expected
                Error           :   BOOL;                       //  Signals that an error has occurred within the method
                ErrorID         :   DINT;                       //  Error identification
                HomeAbsSwitch   :   BOOL;                       //  Digital home switch input is active
                LimitSwitchPos  :   BOOL;                       //  Positive hardware end switch is active
                LimitSwitchNeg  :   BOOL;                       //  Negative hardware end switch is active
                Simulation      :   BOOL;                       //  Axis is in simulation mode (e.g. motor is simulated)
                CommunicationReady: BOOL;                       //  “Network” is initialized and ready for communication
                ReadyForPowerOn :   BOOL;                       //  Drive is ready to be enabled (power on)
                PowerOn         :   BOOL;                       //  If TRUE shows that the power stage is switched ON
                IsHomed         :   BOOL;                       //  The absolute reference position is known for the axis (axis is homed)
                AxisWarning     :   BOOL;                       //  Warning(s) on the axis is present
            END_VAR
        END_METHOD

        ///<summary>
        /// This method presents general axis errors not relating to the methods.
        /// (for instance axis errors, drive errors, communication errors)
        /// This vendor specific method must be overridden in the derived class.
        ///<summary>
        METHOD PUBLIC ABSTRACT MC_ReadAxisError
            VAR_INPUT
                AxisRef         :   AXOpen.Components.Abstractions.Drives.IAxoAxisReference;
                Enable          :   BOOL;                       //  Get the value of the parameter continuously while enabled
            END_VAR
            VAR_OUTPUT
                Valid           :   BOOL;                       //  A valid output is available at the method
                Busy            :   BOOL;                       //  The method is not finished and new output values are to be expected
                Error           :   BOOL;                       //  Signals that an error has occurred within the method
                ErrorID         :   DINT;                       //  Error identification
                AxisErrorID     :   DWORD;                      //  The value of the axis error. These values are vendor specific
            END_VAR
        END_METHOD

        ///<summary>
        /// This method makes the transition from the state ‘ErrorStop’ to ‘Standstill’ or ‘Disabled’ by resetting all
        /// internal axis-related errors – it does not affect the output of the other methods.
        /// This vendor specific method must be overridden in the derived class.
        ///<summary>
        METHOD PUBLIC ABSTRACT MC_Reset
            VAR_INPUT
                AxisRef         :   AXOpen.Components.Abstractions.Drives.IAxoAxisReference;
                Execute         :   BOOL;                       //  Resets all internal axis-related error
            END_VAR
            VAR_OUTPUT
                Done            :   BOOL;                       //  ‘Standstill’ or ‘Disabled’ state is reached
                Busy            :   BOOL;                       //  The method is not finished and new output values are to be expected
                Error           :   BOOL;                       //  Signals that an error has occurred within the method
                ErrorID         :   DINT;                       //  Error identification
            END_VAR
        END_METHOD
    END_CLASS
END_NAMESPACE

(* ---- AxoDrive_Config.st ---- *)
NAMESPACE AXOpen.Components.Drives
    {#ix-attr:[Container(Layout.Wrap)]}
    {S7.extern=ReadWrite}
    CLASS AxoDrive_Config
        VAR PUBLIC
            {#ix-set:AttributeName = "<#Info time#>"}
            InfoTime : LTIME := LT#2S;
            {#ix-set:AttributeName = "<#Error time#>"}
            ErrorTime : LTIME := LT#5S;
            {#ix-set:AttributeName = "<#Task timeout#>"}
            TaskTimeout : LTIME := LT#50S;
            {#ix-set:AttributeName = "<#InTorque window percentage#>"}
            InTorqueWindowPerCent     :   LREAL := LREAL#5.0;
            {#ix-set:AttributeName = "<#InTorque window time#>"}
            InTorqueWindowTime     : LTIME := LT#100ms;
            {#ix-set:AttributeName = "<#InPosition window#>"}
            InPositionWindow     :   LREAL := LREAL#0.05;
        END_VAR
    END_CLASS
END_NAMESPACE

(* ---- AxoDrive_Status.st ---- *)
USING AXOpen.Core;
NAMESPACE AXOpen.Components.Drives
    {#ix-attr:[Container(Layout.Stack)]}
    {S7.extern=ReadWrite}
    CLASS AxoDrive_Status EXTENDS AXOpen.Components.Abstractions.AxoComponent_Status
        VAR PUBLIC
            {#ix-attr:[ReadOnly()]}
            CurrentMotionTaskId    :   eAxoMotionTaskId := eAxoMotionTaskId#Axo_None;
        END_VAR
    END_CLASS
END_NAMESPACE

(* ---- AxoDriveParameterChannelIDN.st ---- *)
USING AXOpen.Core;
NAMESPACE AXOpen.Components.Drives
    CLASS AxoDriveParameterChannelIdnIn
        VAR PUBLIC
            StatusWord  :   WORD;
            Index       :   WORD;
            SubIndex    :   WORD;
            ValueHigh   :   WORD;
            ValueLow    :   WORD;
        END_VAR
    END_CLASS
    CLASS AxoDriveParameterChannelIdnOut
        VAR PUBLIC
            ControlWord :   WORD;
            Index       :   WORD;
            SubIndex    :   WORD;
            ValueHigh   :   WORD;
            ValueLow    :   WORD;
        END_VAR
    END_CLASS
END_NAMESPACE

(* ---- AxoMotionJogTask.st ---- *)
USING AXOpen.Core;

NAMESPACE AXOpen.Components.Drives
    CLASS PUBLIC AxoMotionJogTask EXTENDS AXOpen.Core.AxoMomentaryTask
        VAR PUBLIC
            StartMotion :   BOOL;
            StopMotion  :   BOOL;
        END_VAR
        METHOD PROTECTED OVERRIDE OnSwitchedOn
            StartMotion :=  TRUE;
            StopMotion  :=  FALSE;
        END_METHOD
        METHOD PROTECTED OVERRIDE OnSwitchedOff
            StartMotion :=  FALSE;
            StopMotion  :=  TRUE;
        END_METHOD
    END_CLASS
END_NAMESPACE
